FUNCTION TFPalletizerModulesCheckPowerActive : BOOL (* Funzione che ritorna TRUE se tutti gli assi sono in Power *)
VAR_INPUT
	Modules : POINTER TO TFPalletizerModules;
END_VAR
VAR
END_VAR

TFPalletizerModulesCheckPowerActive:=	
								 (Modules^.AX_X.Ax^.Status.PowerActive OR (Modules^.AX_X.Ax^.BrakeEnable AND Modules^.AX_X.Ax^.BrakePresent))AND
								 (Modules^.AX_Y.Ax^.Status.PowerActive OR (Modules^.AX_Y.Ax^.BrakeEnable AND Modules^.AX_Y.Ax^.BrakePresent))AND
								 (Modules^.AX_Z.Ax^.Status.PowerActive OR (Modules^.AX_Z.Ax^.BrakeEnable AND Modules^.AX_Z.Ax^.BrakePresent))AND
								 (Modules^.AX_J.Ax^.Status.PowerActive OR (Modules^.AX_J.Ax^.BrakeEnable AND Modules^.AX_J.Ax^.BrakePresent));

END_FUNCTION

(* stored: Version 1.1.0.1, ProductVersion 3.1.4024.11
   POU TFPalletizerModulesCheckPowerActive: Id {835a485e-c21e-4625-a4ac-436ce06348e9}, SpecialFunc None *)
